{attribute 'linkalways'}
{attribute 'no_explicit_call' := 'This FB is a CLASS and must be accessed using methods or properties'}
{attribute 'enable_dynamic_creation'}
FUNCTION_BLOCK _ETcVnMergeRegionsOptions EXTENDS EnumDatatypeBase
VAR
	localData : ETcVnMergeRegionsOptions;
	activeData : REFERENCE TO ETcVnMergeRegionsOptions;
	enumBaseDatatype : _ULINT(localData);
END_VAR

METHOD PRIVATE AddLocalEnumeration
VAR_INPUT
	Enumeration : T_MAXSTRING;
	Value : ETcVnMergeRegionsOptions;
END_VAR
AddEnumeration(Enumeration, Value);
END_METHOD

PROPERTY PUBLIC Address : PVOID
GET
Address := ADR(activeData);
END_GET
END_PROPERTY

METHOD PUBLIC ClearReference
VAR_INPUT
END_VAR
activeData REF= localData;
SetBaseDatatypeReference();
END_METHOD

METHOD PUBLIC Clone : I_Datatype
VAR
    pClone : POINTER TO _ETcVnMergeRegionsOptions;
END_VAR
pClone := __NEW(_ETcVnMergeRegionsOptions(InitialValue := Value));
IF pClone = 0 THEN
    RETURN;
END_IF
Clone := pClone^;
END_METHOD

METHOD FB_init : BOOL
VAR_INPUT
	bInitRetains : BOOL; // if TRUE, the retain variables are initialized (warm start / cold start)
	bInCopyCode : BOOL;  // if TRUE, the instance afterwards gets moved into the copy code (online change)
	InitialValue : ETcVnMergeRegionsOptions;
END_VAR
localData := InitialValue;
AddBaseDatatype(enumBaseDatatype);
ClearReference();

AddLocalEnumeration('TCVN_MRO_UPRIGHTBOUNDINGRECT', ETcVnMergeRegionsOptions.TCVN_MRO_UPRIGHTBOUNDINGRECT);
END_METHOD

PROPERTY PUBLIC Identifier : T_MAXSTRING
GET
Identifier := 'ETcVnMergeRegionsOptions';
END_GET
END_PROPERTY

METHOD IsEnumeratorValueEqual : BOOL
VAR_INPUT
	Enumerator : I_KeyValueForwardEnumerator;
END_VAR
VAR
	storedValue : ETcVnMergeRegionsOptions;
END_VAR
IF NOT Enumerator.TryGet(storedValue) THEN
	RETURN;
END_IF

IsEnumeratorValueEqual := storedValue = activeData;
END_METHOD

METHOD PUBLIC MakeReferenceTo
VAR_INPUT
	ReferenceTarget : REFERENCE TO ETcVnMergeRegionsOptions;
END_VAR
activeData REF= ReferenceTarget;
SetBaseDatatypeReference();
END_METHOD

METHOD PROTECTED SetBaseDatatypeReference
VAR_INPUT
END_VAR
enumBaseDatatype.MakeReferenceTo(activeData);
END_METHOD

PROPERTY PUBLIC Size : UDINT
GET
Size := SIZEOF(activeData);
END_GET
END_PROPERTY

METHOD TryMakeReferenceTo : BOOL
VAR_INPUT
	Target : I_Datatype;
END_VAR
VAR
	pTargetData : POINTER TO ETcVnMergeRegionsOptions;
END_VAR
IF NOT IsEquivalentTo(Target) THEN
	RETURN;
END_IF

pTargetData := Target.Address;
activeData REF= pTargetData^;
SetBaseDatatypeReference();
TryMakeReferenceTo := TRUE;
END_METHOD

PROPERTY PUBLIC Value : ETcVnMergeRegionsOptions
GET
Value := activeData;
END_GET
SET
activeData := Value;
END_SET
END_PROPERTY

END_FUNCTION_BLOCK

(* stored: Version 1.1.0.1, ProductVersion 3.1.4026.13
   POU _ETcVnMergeRegionsOptions: Id {02831754-ed06-4090-8059-2e84a007d745}, SpecialFunc None
   Folder Core: Id {045618a8-bbea-499e-9f31-559155afc200}
   Folder Protected: Id {f079924a-0068-442d-9bef-5a99a6e2261c}
   Folder Customize: Id {50de1d73-6796-43ca-bc21-05d0481d0473}
   Folder Constructor: Id {2e7aa681-3f28-49ae-9213-cc333ca68f6e}
   Folder Private: Id {4b5c3495-97ca-44e0-82ee-d626e50b76f1}
   Folder Protected: Id {2c6d00d2-fed1-47fe-a321-4e01552a72e2}
   Method AddLocalEnumeration: Id {f0877e57-2d59-4f5f-9bfa-0d94ab9e8c22}
   Property Address: Id {1115865b-6f4d-4a32-8b8d-f0c9cd5c9f7c}
   Get Get: Id {08a7327a-5861-449d-9b1e-a4b59021daf2}
   Method ClearReference: Id {25a56419-91de-42de-bf4d-abf66f23b4b0}
   Method Clone: Id {9ccb9067-22f0-478a-9b35-6d7f3b71cc03}
   Method FB_init: Id {03fabe17-9dae-4e2a-a0fa-b64327019be4}
   Property Identifier: Id {07242cf8-9c5d-4267-9fc5-1674275ba86d}
   Get Get: Id {d863edbc-84cd-4ade-9775-ac6c466d3681}
   Method IsEnumeratorValueEqual: Id {b66af932-7e04-45cf-85b9-2b12458857d1}
   Method MakeReferenceTo: Id {944a7783-6da3-4888-9c6b-6ba203cf79de}
   Method SetBaseDatatypeReference: Id {1605942b-a3e2-4169-a723-91608a85c2ec}
   Property Size: Id {ee91afc7-04bb-48f5-81ab-dece01ba46a1}
   Get Get: Id {bdd0ad09-3b98-4873-8940-5318582f3916}
   Method TryMakeReferenceTo: Id {f2eb8d0f-32d0-431e-aa94-319a42f01f56}
   Property Value: Id {3774bd3e-d223-4cdd-8a08-65bfe7195dcd}
   Get Get: Id {a8188445-3ec0-4c87-9b5b-a57158671c2b}
   Set Set: Id {0f03f972-fbaa-4121-ab8d-5be041bc76f8} *)
